(* Logix 5000 project; controller WWTP_SEC_CLX vendor 1 type 14 code 54 rev 17.2; software revision 17.00; part 13 of 13 *)
(* tags used below, declared in another part *)
   I_SecTk02_InAuto : ALIAS FOR Local:2:I.DATA.7;
   I_SecTk02_InAuto_IOFault : ALIAS FOR Local:2:I.Fault.7;
   I_SecTk02_RunFdbk : ALIAS FOR Local:2:I.DATA.6;
   I_SecTk02_RunFdbk_IOFault : ALIAS FOR Local:2:I.Fault.6;
   I_SecTk02_Torque : ALIAS FOR Local:2:I.DATA.8;
   I_SecTk02_Torque_IOFault : ALIAS FOR Local:2:I.Fault.8;
   O_SecTk02_Out_Run : ALIAS FOR Local:4:O.DATA.1;   // Secondary Tank #2 Start/Stop
   PLC_Device_ResetPB : BOOL;   // Site Wide Device Reset Push Button
   PLC_Simulation : BOOL;   // Application running IN SIMULATION
(* SecTank01_RAS_Pump, continued *)

ROUTINE Main   (* ladder *)
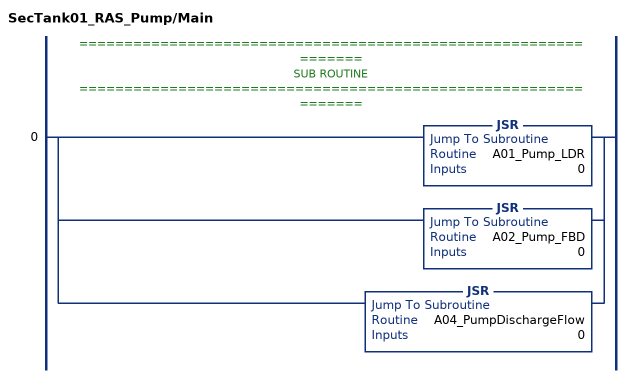
   // ===============================================================
   // SUB ROUTINE
   // ===============================================================
   0: [JSR(A01_Pump_LDR,0) ,JSR(A02_Pump_FBD,0) ,JSR(A04_PumpDischargeFlow,0) ];
END_ROUTINE
END_PROGRAM

PROGRAM SecTank02_Drive   (* main routine Main *)
VAR
   Equip_GroupReset : ALIAS FOR PLC_Device_ResetPB;
   Equip_InAuto : ALIAS FOR I_SecTk02_InAuto;
   Equip_InAuto_IOFault : ALIAS FOR I_SecTk02_InAuto_IOFault;
   Equip_Intlk : ALIAS FOR SecTk02_Intlk;
   Equip_IOFault : BOOL;
   Equip_Motor : ALIAS FOR SecTk02_Motor;
   Equip_Out_Run : ALIAS FOR O_SecTk02_Out_Run;
   Equip_RunFdbk : ALIAS FOR I_SecTk02_RunFdbk;
   Equip_RunFdbk_IOFault : ALIAS FOR I_SecTk02_RunFdbk_IOFault;
   Equip_Torque : ALIAS FOR I_SecTk02_Torque;
   Equip_Torque_IOFault : ALIAS FOR I_SecTk02_Torque_IOFault;
   Wrk_Hand : BOOL;
   Wrk_ResetReqd : BOOL;
   Wrk_ResetRequired : BOOL;
END_VAR

ROUTINE A01_Drive_LDR   (* ladder *)
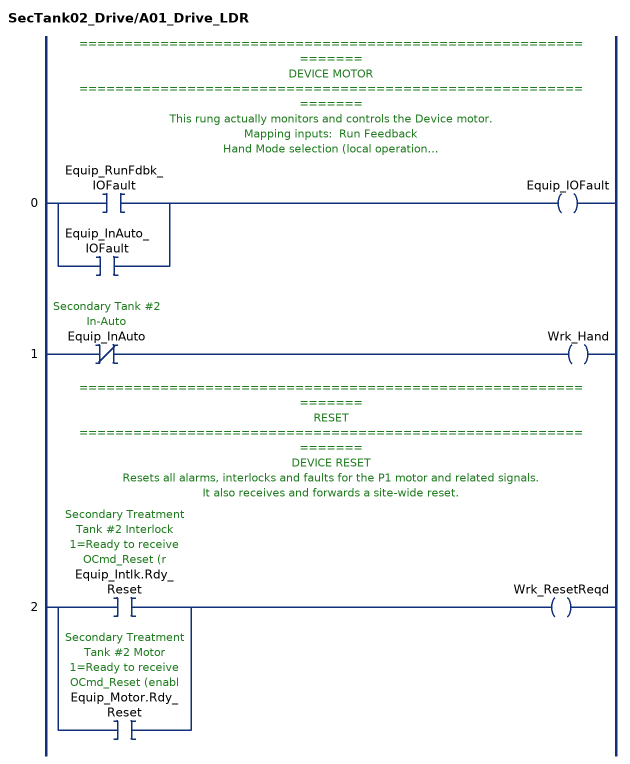
   // ===============================================================
   // DEVICE MOTOR
   // ===============================================================
   // This rung actually monitors and controls the Device motor.
   // Mapping inputs:  Run Feedback
   // Hand Mode selection (local operation)
   // Permissive OK
   // Protective’s OK,
   // I/O Fault signals
   // Pump Reset (above)
   // DEVICE
   // Output Mapping: Starter output
   0: [XIC(Equip_RunFdbk_IOFault) ,XIC(Equip_InAuto_IOFault) ]OTE(Equip_IOFault);
   1: XIO(Equip_InAuto)OTE(Wrk_Hand);
   // ===============================================================
   // RESET
   // ===============================================================
   // DEVICE RESET
   // Resets all alarms, interlocks and faults for the P1 motor and related signals.
   // It also receives and forwards a site-wide reset.
   2: [XIC(Equip_Intlk.Rdy_Reset) ,XIC(Equip_Motor.Rdy_Reset) ]OTE(Wrk_ResetReqd);
END_ROUTINE

ROUTINE A02_Drive_FBD   (* function block diagram *)
   SHEET 1   // Motor
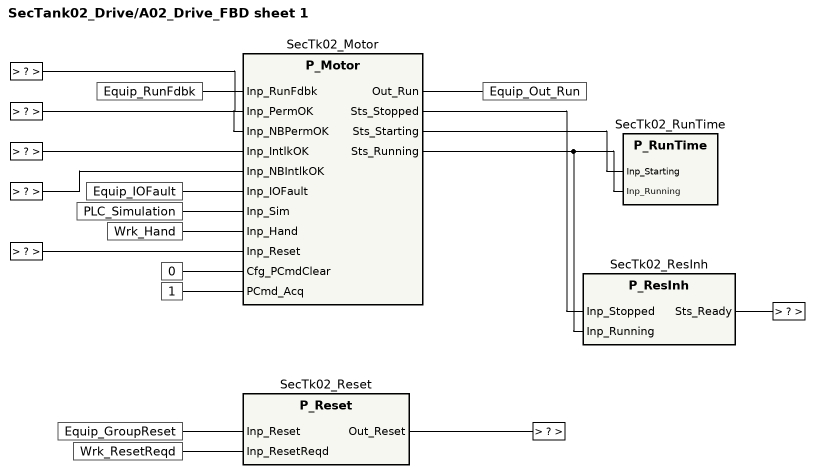
   SecTk02_Reset : P_Reset(Inp_Reset := Equip_GroupReset, Inp_ResetReqd := Wrk_ResetReqd);
   WIRE(?) := SecTk02_Reset.Out_Reset;
   SecTk02_ResInh : P_ResInh(Inp_Stopped := SecTk02_Motor.Sts_Stopped {feedback}, Inp_Running := SecTk02_Motor.Sts_Running {feedback});
   WIRE(?) := SecTk02_ResInh.Sts_Ready;
   SecTk02_Motor : P_Motor(Inp_RunFdbk := Equip_RunFdbk, Inp_PermOK := WIRE(?), Inp_NBPermOK := WIRE(?), Inp_IntlkOK := WIRE(?), Inp_NBIntlkOK := WIRE(?), Inp_IOFault := Equip_IOFault, Inp_Sim := PLC_Simulation, Inp_Hand := Wrk_Hand, Inp_Reset := WIRE(?), Cfg_PCmdClear := 0, PCmd_Acq := 1);
   Equip_Out_Run := SecTk02_Motor.Out_Run;
   SecTk02_RunTime : P_RunTime(Inp_Starting := SecTk02_Motor.Sts_Starting, Inp_Running := SecTk02_Motor.Sts_Running);
   SHEET 2   // Permissives
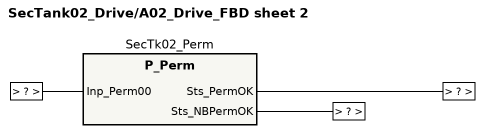
   SecTk02_Perm : P_Perm(Inp_Perm00 := WIRE(?));
   WIRE(?) := SecTk02_Perm.Sts_NBPermOK;
   WIRE(?) := SecTk02_Perm.Sts_PermOK;
   SHEET 3   // Interlocks
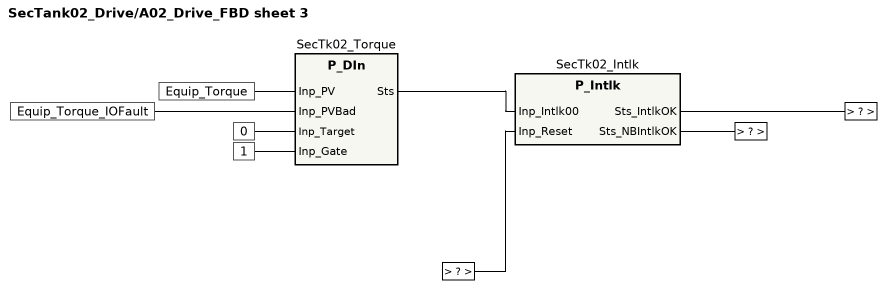
   SecTk02_Torque : P_DIn(Inp_PV := Equip_Torque, Inp_PVBad := Equip_Torque_IOFault, Inp_Target := 0, Inp_Gate := 1);
   SecTk02_Intlk : P_Intlk(Inp_Intlk00 := SecTk02_Torque.Sts, Inp_Reset := WIRE(?));
   WIRE(?) := SecTk02_Intlk.Sts_NBIntlkOK;
   WIRE(?) := SecTk02_Intlk.Sts_IntlkOK;
END_ROUTINE

ROUTINE Main   (* ladder *)
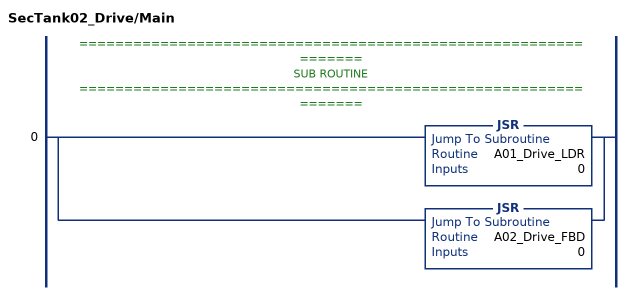
   // ===============================================================
   // SUB ROUTINE
   // ===============================================================
   0: [JSR(A01_Drive_LDR,0) ,JSR(A02_Drive_FBD,0) ];
END_ROUTINE
END_PROGRAM
